ADAPTER ASR_AX (* bidirectional Adapter Interface for 2 Events (forward, Set/Reset) and 1 Bool (backward, AX-style) *)
  (* Standard: 61499-1; Description: Copyright (c) 2026 HR Agrartechnik GmbH This program and the accompanying materials are made available under the terms of the Eclipse Public License 2.0 which is available at https://www.eclipse.org/legal/epl-2.0/ SPDX-License-Identifier: EPL-2.0 *)
  (* Version 1.0, 2026-09-03, Franz Höpfinger, HR Agrartechnik GmbH, Initial Version *)
  PACKAGE adapter::types::bidirectional;
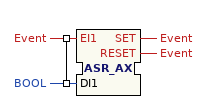
  EVENT_INPUT
    EI1 WITH DI1; (* Indication (or Request) *)
  END_EVENT
  EVENT_OUTPUT
    SET; (* Set / Switch on *)
    RESET; (* Reset / Switch off *)
  END_EVENT
  VAR_INPUT
    DI1 : BOOL; (* Indication (or Request) Data to Plug *)
  END_VAR
END_ADAPTER
